(* PLC project Generated.project, CODESYS CODESYS V3.5 SP19 Patch 1 *)
(* stored: creationDateTime 2026-11-18T10:35:01.105488, modificationDateTime 2026-11-18T10:35:01.105488 *)

(* ═══════════════════════════════════════════════════════════════ 🌐 ST_CommunHMI — Données d'échange IHM COMMUNES (pas propres à un axe) ─────────────────────────────────────────────────────────────── Regroupe les signaux qui ne concernent PAS un axe/mécanisme en particulier (1 seul capteur/signal partagé par toute la machine) — évite de les dupliquer ou de les laisser en variables isolées directement dans GVL_IHM. Exemple : TopPositionSensorActive (capteur unique, commun M1+M2), BrakeThermalFault (retour unique, commun M1+M2+M3). ⚠️ Ne pas y mettre HmiInitDone (indicateur interne de séquencement boot, pas une information machine destinée à l'opérateur) — reste seul dans GVL_IHM. 🧭 Structuration homogène : états → Cfg → Bypass (Cfg au-dessus de Bypass, Bypass en bas), cohérent avec ST_WinchHMI / ST_SyncHMI. ═══════════════════════════════════════════════════════════════ *)
TYPE ST_CommunHMI : STRUCT
  TopPositionSensorActive : BOOL;  (* ⚠️ Capteur de position haute commun M1+M2 détecté *)
  TopHardStopLatched : BOOL;  (* 🔒 Latch directionnel capteur position haute commun M1+M2 actif *)
  BrakeThermalFault : BOOL;  (* 🌡️ Défaut/perte thermique frein — retour unique commun M1/M2/M3, escalade PowerCutOff *)
  PhaseRotationFault : BOOL;  (* ⚡ Rotation de phase incorrecte — retour unique commun M1/M2/M3 *)
  LimitLegalReached : BOOL;  (* 📐 Limite légale de profondeur de dragage atteinte (globale) *)
  HydraulicThermalFault : BOOL;  (* 🌡️ Défaut/perte thermique centrale hydraulique *)
  SimTopSensorBypassActive : BOOL;  (* 🩺 Indicateurs diagnostic bypass — PLC→IHM, état réellement consommé 🩺 1 = Bypass.TopLimitSwitch réellement actif *)
  SimSlackCableBypassActive : BOOL;  (* 🩺 1 = Bypass.SlackCable réellement actif *)
  WinchInputSourceChanged : BOOL;  (* 🔀 PLC→IHM : source Winch a basculé (réel/simu) ce cycle *)
  TglHeartbeatIhm : BOOL;  (* 💓 Heartbeat IHM↔PLC — IHM inverse TglHeartbeatIhm toutes les 500 ms. IHM→PLC : toggle périodique, jamais valeur constante *)
  TglHeartbeatPlc : BOOL;  (* PLC→IHM : clignotant activité PLC *)
  HeartbeatIhmOk : BOOL;  (* PLC→IHM : front IHM post-boot reçu et timeout absent *)
  HeartbeatIhmTimeout : BOOL;  (* PLC→IHM : aucun front IHM depuis 2 s *)
  HeartbeatIhmElapsed : TIME;  (* PLC→IHM : temps depuis dernier front IHM *)
  BtnWinchBothAscent : BOOL;  (* Boutons pilotage direct des 2 treuils (communs, remplace SelJoystickWinch en mode boutons) ⬆️ Monte les 2 treuils simultanément *)
  BtnWinchBothDescent : BOOL;  (* ⬇️ Descend les 2 treuils simultanément *)
  ConfigRestoredFromPersistent : BOOL;  (* Alarme restauration config PERSISTENT (RETAIN invalidé, ex. changement de struct ST_*HMI) — visible et acquittable, jamais de disparition automatique silencieuse (doctrine reset=front, PRG_07_Supervision.st §2bis). Vérifier les valeurs avant reprise cycle. ⚠️ PLC→IHM : restauration détectée ce boot, à vérifier *)
  BtnAckConfigRestored : BOOL;  (* 🔘 IHM→PLC : acquittement opérateur (front) *)
  Preflight : ST_PreflightHMI;  (* 🩺 Verdict observateur à l'arrêt — jamais bloquant *)
  WinchSymmetry : ST_WinchSymmetryHMI;  (* ⚖️ Mesures passives M1/M2 *)
  KoboldImmersionConfirmed : BOOL;  (* 🩺 Diagnostic arrêt auto descente Kobold (pilotage normal) Front Kobold confirmé dans la fenêtre d'immersion *)
  KoboldBottomTouchLatched : BOOL;  (* Fond détecté, descente bloquée (ProcessPermitM1/M2_Descend) *)
  RunningHours : ST_RunningHoursHMI;  (* ⏱️ Compteurs horaires maintenance — Machine (PLC sous tension) + M1/M2/M3 (marche reelle) *)
  EncoderCfg : ST_fbEncoder_Cfg;  (* ⚙️ Configuration technologique codeur commune M1/M2 Réglage mode confirmation preset, ponté vers GVL_PERSISTENT *)
  Cfg : ST_CommunCfg;  (* 📐 Configuration des paramètres communs machine (au-dessus des bypass) *)
  Bypass : ST_BypassCommun;  (* 🔒 Bypass maintenance de capteurs COMMUNS (voir REGISTRE_ACTIONS_Bypass_v1.0 (archive)) 🔒 Granulaire, applique le bypass aux 2 treuils simultanément (pilotage "both") — OR avec le bypass individuel M1/M2 dans PRG_04 *)
END_STRUCT;
END_TYPE

(* ═══════════════════════════════════════════════════════════════ ST_BypassCommun — Bypass maintenance GRANULAIRE, applicable aux 2 treuils à la fois ─────────────────────────────────────────────────────────────── 🎨 Distinct des bypass individuels M1/M2 (ST_BypassWinch) un OUI ici lève la protection sur LES DEUX treuils simultanément (pilotage "both", GVL_IHM.Commun.BtnWinchBothAscent/Descent), en OR avec le bypass individuel de chaque instance (PRG_04_Treuils_Benne). Évite de devoir activer 2 fois le même bypass (M1 ET M2) avant un pilotage groupé — SANS retirer les bypass individuels pour le pilotage à l'unité. ⚠️ Ne remplace PAS les bypass individuels : les deux se combinent en OR, jamais l'un n'entraîne la désactivation de l'autre. 🔒 Doctrine : actionnable UNIQUEMENT en MAINT_N2, RETAIN, jamais masque les autres défauts du même bloc (voir REGISTRE_ACTIONS_Bypass_v1.0 (archive)). ═══════════════════════════════════════════════════════════════ *)
TYPE ST_BypassCommun : STRUCT
  Global : BOOL;  (* 🌐 Bypass Global Commun (toutes sécurités communes M1+M2) *)
  SlackCable : BOOL;  (* ⚠️ Bypass capteur mou de câble — capteur unique M1/M2, OR avec bypass individuel *)
  TopLimitSwitch : BOOL;  (* 🚧 Bypass fin de course physique haute (capteur, bit5), OR avec bypass individuel *)
  TopLimitSoftware : BOOL;  (* : Bypass fin de course logiciel haut (position calculée), OR avec bypass individuel *)
  CableLimitSwitch : BOOL;  (* : Bypass limite basse physique (longueur câble), OR avec bypass individuel *)
  LimitLegal : BOOL;  (* : Bypass limite légale de profondeur, OR avec bypass individuel *)
  Initialized : BOOL;  (* Initialisé au boot *)
END_STRUCT;
END_TYPE

(* ═══════════════════════════════════════════════════════════════ ST_CommunCfg — Configuration des paramètres communs machine ═══════════════════════════════════════════════════════════════ *)
TYPE ST_CommunCfg : STRUCT
  LimitLegalDepthMinAllowed_M : REAL := -30;  (* Blocage instantané à 0m : sans défaut explicite, ce champ vaut 0.0 tant qu'il n'a pas été réglé côté IHM -- "CablePosM <= 0.0" se déclenche dès la position de référence, avant tout réglage réel de la cote légale. Défaut -999.0 (jamais atteint en pratique) : LimitLegalEnabled=TRUE sans réglage ne bloque plus rien par erreur -- il faut régler la vraie cote pour que la protection devienne active. 📐 Cote min de dragage autorisée (m, négatif) *)
  LimitLegalEnabled : BOOL;  (* 🟢 Activation de la limite légale *)
  SelHomingApproachEnable : BOOL;  (* 🔌 Case IHM : autorise le dépassement butée haute pour homing (si MAINT_N2) *)
  WinchMaxStepDescent : INT := 5;  (* 🚀 Plafond palier descente nominal (1..5), commun M1/M2 *)
  WinchMaxStepAscent : INT := 5;  (* 🚀 Limitation palier vitesse en montée (1..5), commun M1/M2 *)
  WinchSlowdownDistanceTop_M : REAL := 0.5;  (* 📏 Distance avant limite haute : 0 = arrêt au seuil (m), commun M1/M2 *)
  WinchSlowdownDistanceBottom_M : REAL := 1;  (* 📏 Distance avant limite basse pour ralentir (m), commun M1/M2 *)
  WinchSlowdownMaxStep : INT := 1;  (* : WinchSlowSpeed_Pct (%) retiré — un treuil ne connaît que des paliers (1..5), pas une vitesse continue. : Plafond palier dans la zone de ralentissement (1..5), commun M1/M2 *)
  CfgCableLimitAscent_M : REAL := 7.5;  (* 📐 Limite haute d'exploitation NORMALE (m), commun M1/M2 *)
  TglEnableKoboldAutoStopDescent : BOOL := FALSE;  (* : Arrêt auto descente sur détection fond Kobold (pilotage normal) *)
  TglEnableCoupledBucketSequencing : BOOL := TRUE;  (* Séquencement auto benne en pilotage couplé (WinchSel=0, MAINT_N1/N2) : pousser le joystick benne pas ouverte -> ouvre d'abord puis descend couplé ; tirer benne pas fermée -> ferme d'abord puis remonte couplé. Défaut TRUE (activé) ; 1 bouton IHM pour désactiver -> comportement brut (2 treuils sans condition). OFF = jamais gouverné par instBucket.Busy hors action MANUELLE benne (WinchSel=2) / DumpAtTremie / ExtractionAssist. *)
  TglEnableWinchDescentLock_M3 : BOOL := TRUE;  (* 🔒 Verrouillage descente treuil M1/M2 en mode MAINT si le pont M3 n'est pas à P1/Maintenance : Défaut TRUE (sécurisé) ; bouton IHM pour désactiver (permet descente treuils partout). *)
  Initialized : BOOL := FALSE;  (* 🚦 flag restauration boot *)
END_STRUCT;
END_TYPE

TYPE ST_PreflightHMI : STRUCT
  BtnRun : BOOL;
  PreflightOk : BOOL;
  PreflightDone : BOOL;
  PreflightBusy : BOOL;
  PreflightErrorId : WORD;
END_STRUCT;
END_TYPE

(* ═══════════════════════════════════════════════════════════════ ⏱️ ST_RunningHoursHMI — Compteurs horaires maintenance (PLC→IHM) ─────────────────────────────────────────────────────────────── 🎯 Role : totalisateurs de marche pour planification maintenance, independants du chrono de cycle (qui se remet a zero par passe). 🔌 Machine = duree sous tension PLC (toujours active des le boot). M1/M2/M3 = duree contacteur marche reel actif (preuve physique). 💾 Source RETAIN : GVL_PERSISTENT (secondes), converties ici en H:Min. ═══════════════════════════════════════════════════════════════ *)
TYPE ST_RunningHoursHMI : STRUCT
  MachineHours_H : DINT;  (* Heures entieres, PLC sous tension *)
  MachineHours_Min : INT;  (* Minutes 0..59 *)
  M1Hours_H : DINT;  (* Heures entieres, treuil M1 en marche *)
  M1Hours_Min : INT;
  M2Hours_H : DINT;  (* Heures entieres, treuil M2 en marche *)
  M2Hours_Min : INT;
  M3Hours_H : DINT;  (* Heures entieres, translation M3 en marche *)
  M3Hours_Min : INT;
END_STRUCT;
END_TYPE

TYPE ST_WinchSymmetryHMI : STRUCT
  BtnReset : BOOL;
  SymmetryOk : BOOL;
  SymmetryValid : BOOL;
  DeltaStartDelay_Ms : UDINT;
  DeltaBrakeReleaseTime_Ms : UDINT;
  DeltaBrakeApplyTime_Ms : UDINT;
  DeltaStopDistance_M : REAL;
  DeltaStopTime_Ms : UDINT;
  MaxSyncDeviation_M : REAL;
END_STRUCT;
END_TYPE

(* ======================================================================= ⚙️ ST_fbEncoder_Cfg — Réglages technologiques publics de FB_Encoder ─────────────────────────────────────────────────────────────────────── 🎯 Rôle : porter le mode de confirmation preset commun aux codeurs. 🔒 Ownership : GVL_IHM.Commun.EncoderCfg ↔ GVL_PERSISTENT._EncoderCfgPersist. 📄 Doc : DOC/AF/AF_Partie-09_Fonction_Encoder_v2.4.md ======================================================================= *)
TYPE ST_fbEncoder_Cfg : STRUCT
  PresetConfirmMode : E_PresetConfirmMode := E_PresetConfirmMode.READBACK_ONLY;  (* Mode de confirmation preset, défaut relecture *)
  Initialized : BOOL := FALSE;  (* 🚦 TRUE après restauration du pont persistant *)
END_STRUCT;
END_TYPE

(* values of E_PresetConfirmMode: READBACK_ONLY: Confirmation par relecture de position; READBACK_AND_STATUSBIT: Relecture et bit d'état matériel; STATUSBIT_ONLY: Bit d'état matériel uniquement *)

{attribute 'qualified_only'}
{attribute 'strict'}
TYPE E_PresetConfirmMode : (READBACK_ONLY := 0, READBACK_AND_STATUSBIT := 1, STATUSBIT_ONLY := 2);
END_TYPE
